(* CODESYS project testIO.project

Project tree, tasks and I/O mapping:
  Device : Jinan Cherry-ARM Cortex-VxWorks, Jinan Cheery Electric Co., Ltd., version 3.5.11.20
    application Application
      libraries: Standard, * (System)
      task MainTask (cyclic, interval 500 ms, priority 1) calls PLC_PRG
      program PLC_PRG [ST]
    SoftMotion General Axis Pool
    IoDrvSOC : IoDrvSOC, Hitech, version 1.0.0.0
        input  Application.PLC_PRG.sDI[1] : BOOL  // in1
        input  Application.PLC_PRG.sDI[2] : BOOL  // in2
        input  Application.PLC_PRG.sDI[3] : BOOL  // in6
        input  Application.PLC_PRG.sDI[4] : BOOL  // in7
        input  Application.PLC_PRG.sDI[5] : BOOL  // in8
        output Application.PLC_PRG.sDO[1] : BOOL  // out1
        output Application.PLC_PRG.sDO[2] : BOOL  // out2
        output Application.PLC_PRG.sDO[3] : BOOL  // out3
        output Application.PLC_PRG.sDO[4] : BOOL  // out4
        output Application.PLC_PRG.sDO[5] : BOOL  // out5
        unmapped channels: in3, in4, in5, out6, out7, out8
*)

// Device/Application/PLC_PRG
PROGRAM PLC_PRG
VAR
	sDO : ARRAY[1..5] OF BOOL;
	sDI : ARRAY[1..5] OF BOOL;
	i : INT;
	init : BOOL;
END_VAR

IF init = FALSE THEN
	FOR i := 1 TO 5 BY +1 DO
		sDO[i] := 1;
		sDI[i] := 0;
	END_FOR
	init := TRUE;
END_IF

END_PROGRAM
